// TIA Portal V19 export
VAR_GLOBAL   // PLC tag table "Diagnostics"
END_VAR
VAR_GLOBAL CONSTANT   // user constants
   NO_OF_EM : UDInt := 16;   // Highest value of EMs
END_VAR
